PROGRAM POU
VAR
	eState : E_State;
	VoltMonBd_0: VoltTranBd;
END_VAR

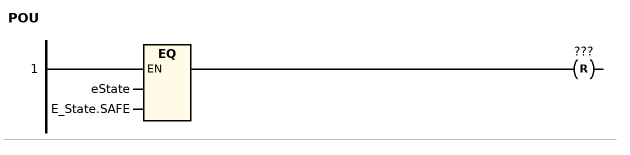
// NETWORK 1
??? R= eState = E_State.SAFE;

END_PROGRAM

(* stored: Version 1.1.0.1, ProductVersion 3.1.4024.11
   POU POU: Id {29d9239d-0139-40b8-9dbf-540e40d8f6a4}, SpecialFunc None *)
